// TIA Portal V16 export
// export: Created 2024-09-05T17:39:13.7356852Z, ExportSetting WithDefaults, DisplayName Totally Integrated Automation Portal, DisplayVersion V16 Update 6, DisplayName TIA Portal Version Control Interface, DisplayVersion V16 Update 2, DisplayName TIA Portal Openness, DisplayVersion V16 Update 6, DisplayName STEP 7 Professional, DisplayVersion V16 Update 6, DisplayName STEP 7 Safety, DisplayVersion V16, DisplayName WinCC Advanced, DisplayVersion V16 Update 6
DATA_BLOCK "READER_SIDE_RH"   // DB70
VERSION : 0.1
// stored: AutoNumber true, DBAccessibleFromOPCUA true, InstanceOfName READER_LOGIC, InstanceOfType FB
"READER_LOGIC"
   // VAR_INPUT
   //    MODE : UInt;
   //    INIT_SCAN : Bool;
   //    SCAN_BUSY : Bool;
   //    SCAN_COMPLETE : Bool;
   //    STA_REC_1 : Bool;
   //    STA_REC : Bool;
   //    SCAN_OK1 : Bool;
   //    SCAN_OK2 : Bool;
   //    IJC_DISABLE : Bool;
   //    SCAN_LABEL : String;
   //    SCAN_POSITION : Int;
   //    SCAN_LEN : Int;
   //    READ_OF_SCAN : HW_SUBMODULE;
   //    NUM_OF_TUBE : Bool;
   //    RESET_SCANER : Bool;
   // END_VAR
   // VAR_OUTPUT
   //    REQUEST_SCAN : Bool;
   //    READ_STRG : String;
   //    SCAN_OK : Bool;
   //    MSG_STATUS_REQ : Bool;
   //    NFP_AUX : String;
   //    LECTURA_SCANER_ST : String;
   //    SCAN_CLEAR : Bool;
   // END_VAR
   // VAR
   //    RET_TRIG : IEC_TIMER;
   // END_VAR
BEGIN
END_DATA_BLOCK
